// TIA Portal V16 export
// export: Created 2021-05-25T16:14:40.4761785Z, ExportSetting WithDefaults, DisplayName Totally Integrated Automation Portal, DisplayVersion V16, DisplayName TIA Portal Version Control Interface, DisplayVersion V16, DisplayName TIA Portal Openness, DisplayVersion V16, DisplayName STEP 7 Professional, DisplayVersion V16, DisplayName STEP 7 Safety, DisplayVersion V16, DisplayName WinCC Unified SCADA Engineering System, DisplayVersion V16
DATA_BLOCK "dbHSC"   // DB37
{ S7_Optimized_Access := 'TRUE'; DB_Accessible_From_OPC_UA := 'FALSE' }
VERSION : 0.1
// stored: AutoNumber false, DBAccessibleFromOPCUA false
   VAR RETAIN
      ScanLineCounts { S7_SetPoint := 'True'} : "udtHSC";
   END_VAR
BEGIN
   ScanLineCounts.EguValue := 31.3194;
END_DATA_BLOCK
